// TIA Portal V19 export
TYPE "udt_FlyingCarriage_CIn"
   STRUCT
      EnableStopDoorOpeningReq : Bool;
      EnableStopInPhase : Bool := TRUE;
      EnableStopProgrammed : Bool := TRUE;
      StopInactivity : Bool;
      Semiauto : Bool := FALSE;
      MovePermit : Bool := FALSE;
      LeadAxisStandstill : Bool;
      ToolAtRest : Bool;
      ToolAtRestManEmptyng : Bool;
      Exe_PosAbs : Bool;
      Exe_Zero : Bool;
      TorqueRequest : Bool;
      PosAbs_TargetPosAx : LReal;
      PosAbs_Vel : LReal;
      PosAbs_Acc : LReal;
      PosAbs_Dec : LReal;
      PosAbs_Jerk : LReal;
   END_STRUCT;
END_TYPE
